# EPICS substitutions: viocs/substitutions/ch.substitutions
file "db/individual.db" {
    pattern { family, pos }
        { "CH", "01C1" }
        { "CH", "01C2" }
        { "CH", "01C3" }
        { "CH", "01C4" }
        { "CH", "01M1" }
        { "CH", "01M2" }
        { "CH", "02C1" }
        { "CH", "02C2" }
        { "CH", "02C3" }
        { "CH", "02C4" }
        { "CH", "02M1" }
        { "CH", "02M2" }
        { "CH", "03C1" }
        { "CH", "03C2" }
        { "CH", "03C3" }
        { "CH", "03C4" }
        { "CH", "03M1" }
        { "CH", "03M2" }
        { "CH", "04C1" }
        { "CH", "04C2" }
        { "CH", "04C3" }
        { "CH", "04C4" }
        { "CH", "04M1" }
        { "CH", "04M2" }
        { "CH", "05C1" }
        { "CH", "05C2" }
        { "CH", "05C3" }
        { "CH", "05C4" }
        { "CH", "05M1" }
        { "CH", "05M2" }
        { "CH", "06C1" }
        { "CH", "06C2" }
        { "CH", "06C3" }
        { "CH", "06C4" }
        { "CH", "06M1" }
        { "CH", "06M2" }
        { "CH", "07C1" }
        { "CH", "07C2" }
        { "CH", "07C3" }
        { "CH", "07C4" }
        { "CH", "07M1" }
        { "CH", "07M2" }
        { "CH", "08C1" }
        { "CH", "08C2" }
        { "CH", "08C3" }
        { "CH", "08C4" }
        { "CH", "08M1" }
        { "CH", "08M2" }
        { "CH", "09C1" }
        { "CH", "09C2" }
        { "CH", "09C3" }
        { "CH", "09C4" }
        { "CH", "09M1" }
        { "CH", "09M2" }
        { "CH", "10C1" }
        { "CH", "10C2" }
        { "CH", "10C3" }
        { "CH", "10C4" }
        { "CH", "10M1" }
        { "CH", "10M2" }
        { "CH", "11C1" }
        { "CH", "11C2" }
        { "CH", "11C3" }
        { "CH", "11C4" }
        { "CH", "11M1" }
        { "CH", "11M2" }
        { "CH", "12C1" }
        { "CH", "12C2" }
        { "CH", "12C3" }
        { "CH", "12C4" }
        { "CH", "12M1" }
        { "CH", "12M2" }
        { "CH", "13C1" }
        { "CH", "13C2" }
        { "CH", "13C3" }
        { "CH", "13C4" }
        { "CH", "13M1" }
        { "CH", "13M2" }
        { "CH", "14C1" }
        { "CH", "14C2" }
        { "CH", "14C3" }
        { "CH", "14C4" }
        { "CH", "14M1" }
        { "CH", "14M2" }
        { "CH", "15C1" }
        { "CH", "15C2" }
        { "CH", "15C3" }
        { "CH", "15C4" }
        { "CH", "15M1" }
        { "CH", "15M2" }
        { "CH", "16C1" }
        { "CH", "16C2" }
        { "CH", "16C3" }
        { "CH", "16C4" }
        { "CH", "16M1" }
        { "CH", "16M2" }
        { "CH", "17C1" }
        { "CH", "17C2" }
        { "CH", "17C3" }
        { "CH", "17C4" }
        { "CH", "17M1" }
        { "CH", "17M2" }
        { "CH", "18C1" }
        { "CH", "18C2" }
        { "CH", "18C3" }
        { "CH", "18C4" }
        { "CH", "18M1" }
        { "CH", "18M2" }
        { "CH", "19C1" }
        { "CH", "19C2" }
        { "CH", "19C3" }
        { "CH", "19C4" }
        { "CH", "19M1" }
        { "CH", "19M2" }
        { "CH", "20C1" }
        { "CH", "20C2" }
        { "CH", "20C3" }
        { "CH", "20C4" }
        { "CH", "20M1" }
        { "CH", "20M2" }
}
